FUNCTION_BLOCK E_CU (* Event-Driven Up Counter *)
  (* Standard: 61499-1-A.18; Classification: Event-driven blocks; Function: Up-counter *)
  (* Version 0.5, 2018-08-20, JHC, Holobloc Inc, Added ECC documentation. *)
  (* Version 0.4, 2018-08-11, JHC, Holobloc Inc, Added CV comment. *)
  (* Version 0.3, 2009-11-16, JHC, Holobloc Inc, Updated for 61499-1 Ed2. *)
  (* Version 0.2, 2006-09-07, JHC, Holobloc Inc, Changed package to fb.rt.events. *)
  (* Version 0.1, 2001-04-27, JHC, Rockwell Automation, XML version *)
  (* Version 0.0, 1999-01-22, JHC, Rockwell Automation, SRC version *)
  (* Compiler header: package fb.rt.events; *)
  (* Compiler Java Sun JDK 1.7.0 *)
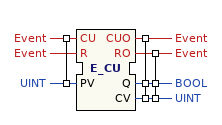
  EVENT_INPUT
    CU WITH PV; (* Count Up *)
    R; (* Reset *)
  END_EVENT
  EVENT_OUTPUT
    CUO WITH Q, CV; (* Count Up Output Event *)
    RO WITH Q, CV; (* Reset Output Event *)
  END_EVENT
  VAR_INPUT
    PV : UINT := 4; (* LImit Value *)
  END_VAR
  VAR_OUTPUT
    Q : BOOL; (* CV >= PV *)
    CV : UINT; (* Current Value *)
  END_VAR
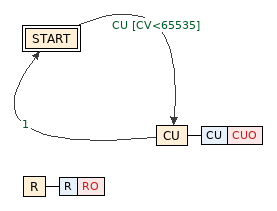
  EC_STATES
    START; (* Initial State *)
    CU : CU -> CUO; (* Count Up *)
    R : R -> RO; (* Service R (Reset) Event *)
  END_STATES
  EC_TRANSITIONS
    START TO CU := CU [CV<65535];
    CU TO START := 1;
  END_TRANSITIONS
  ALGORITHM CU IN ST: (* Count Up *)
CV := CV + 1;
Q := (CV >= PV);
  END_ALGORITHM
  ALGORITHM R IN ST: (* Reset *)
CV := 0;
Q := FALSE;
  END_ALGORITHM
END_FUNCTION_BLOCK
